// TIA Portal V15.1 export
// export: Created 2024-06-21T08:41:11.7725682Z, ExportSetting WithDefaults, DisplayName Totally Integrated Automation Portal, DisplayVersion V15.1 Update 5, DisplayName TIA Portal Openness, DisplayVersion V15.1 Update 5, DisplayName SINAMICS Startdrive Advanced, DisplayVersion V15.1, DisplayName G130, G150, S120, S150, SINAMICS MV, S210, DisplayVersion V15.1, DisplayName G110M, G120, G120C, G120D, G120P, DisplayVersion V15.1, DisplayName STEP 7 Professional, DisplayVersion V15.1 Update 5, DisplayName STEP 7 Safety, DisplayVersion V15.1, DisplayName WinCC Professional, DisplayVersion V15.1 Update 5, DisplayName SIMATIC Visualization Architect, DisplayVersion V15.1
FUNCTION_BLOCK "LGBShiftRegLine"   // FB6704, FBD
TITLE = LGBShiftRegLine
{ S7_Optimized_Access := 'TRUE' }
VERSION : 0.1
// stored: AutoNumber false, IsIECCheckEnabled false, IsRetainMemResEnabled false, MemoryReserve 100, SetENOAutomatically False, UDAEnableTagReadback false
   VAR_INPUT
      I_VEMData { ExternalAccessible := 'False'; ExternalVisible := 'False'; ExternalWritable := 'False'} : "VEMData";   // VEMData
      I_EncPlsCntr { ExternalAccessible := 'False'; ExternalVisible := 'False'; ExternalWritable := 'False'} : DInt;   // Encoder pulse counter - value from counter card
      I_LineRunning { ExternalAccessible := 'False'; ExternalVisible := 'False'; ExternalWritable := 'False'} : Bool;   // Line running - signal from freq. convertor
      I_TriggerDet { ExternalAccessible := 'False'; ExternalVisible := 'False'; ExternalWritable := 'False'} : Bool;   // Trigger sensor
   END_VAR
   VAR_OUTPUT
      O_SetpBodyPitch { ExternalAccessible := 'False'; ExternalVisible := 'False'; ExternalWritable := 'False'} : Int;   // Setpoint Body pitch (cm)
      O_SetpCycleTime { ExternalAccessible := 'False'; ExternalVisible := 'False'; ExternalWritable := 'False'} : Int;   // Setpoint Cycle time (sec)
      O_SetpSpeed { ExternalAccessible := 'False'; ExternalVisible := 'False'; ExternalWritable := 'False'} : Real;   // Setpoint Speed (m/min)
      O_LineIsEmpty { ExternalAccessible := 'False'; ExternalVisible := 'False'; ExternalWritable := 'False'} : Bool;   // Line is empty
      O_Area1 { ExternalAccessible := 'False'; ExternalVisible := 'False'; ExternalWritable := 'False'} : Bool;   // Position active in the Area
      O_Area2 { ExternalAccessible := 'False'; ExternalVisible := 'False'; ExternalWritable := 'False'} : Bool;   // Position active in the Area
      O_Area3 { ExternalAccessible := 'False'; ExternalVisible := 'False'; ExternalWritable := 'False'} : Bool;   // Position active in the Area
      O_Area4 { ExternalAccessible := 'False'; ExternalVisible := 'False'; ExternalWritable := 'False'} : Bool;   // Position active in the Area
      O_Area5 { ExternalAccessible := 'False'; ExternalVisible := 'False'; ExternalWritable := 'False'} : Bool;   // Position active in the Area
      O_Area6 { ExternalAccessible := 'False'; ExternalVisible := 'False'; ExternalWritable := 'False'} : Bool;   // Position active in the Area
      O_Area7 { ExternalAccessible := 'False'; ExternalVisible := 'False'; ExternalWritable := 'False'} : Bool;   // Position active in the Area
      O_Area8 { ExternalAccessible := 'False'; ExternalVisible := 'False'; ExternalWritable := 'False'} : Bool;   // Position active in the Area
      O_Area9 { ExternalAccessible := 'False'; ExternalVisible := 'False'; ExternalWritable := 'False'} : Bool;   // Position active in the Area
      O_Area10 { ExternalAccessible := 'False'; ExternalVisible := 'False'; ExternalWritable := 'False'} : Bool;   // Position active in the Area
      O_AlarmABCondition { ExternalAccessible := 'False'; ExternalVisible := 'False'; ExternalWritable := 'False'} : Bool;   // Alarm AB Condition
      O_AlarmA { ExternalAccessible := 'False'; ExternalVisible := 'False'; ExternalWritable := 'False'} : Bool;   // Alarm A
      O_AlarmB { ExternalAccessible := 'False'; ExternalVisible := 'False'; ExternalWritable := 'False'} : Bool;   // Alarm B
      O_AlarmC { ExternalAccessible := 'False'; ExternalVisible := 'False'; ExternalWritable := 'False'} : Bool;   // Alarm C
      O_AlarmD { ExternalAccessible := 'False'; ExternalVisible := 'False'; ExternalWritable := 'False'} : Bool;   // Alarm D
      H_AlarmDWord { ExternalAccessible := 'False'; ExternalVisible := 'False'; ExternalWritable := 'False'} : DWord;   // Alarm Word
   END_VAR
   VAR_IN_OUT
      IO_ShiftRegData : "ShiftRegData";   // Line data
      IO_Modes : "Modes";   // Modes
      H_HMI : "H_HMI";   // Animation
      H_GBShiftRegLine : "H_GBShiftRegLine";   // Animation
      C_Config : "ShiftRegLineConfig";   // Config
   END_VAR
   VAR
      AA_EncoderMinMax { ExternalAccessible := 'False'; ExternalVisible := 'False'; ExternalWritable := 'False'} : Bool;   // Settings Min. and Max. range for the encoder is not ok --- Max. must be > Min. and Max. <> 0
      AA_SetpointBodyPitch { ExternalAccessible := 'False'; ExternalVisible := 'False'; ExternalWritable := 'False'} : Bool;   // Setpoint Bodypitch is not ok --- Setpoint must be > 100 cm
      AA_SetpointCycleTime { ExternalAccessible := 'False'; ExternalVisible := 'False'; ExternalWritable := 'False'} : Bool;   // Setpoint CycleTime is not ok --- Setpoint must be > 10 sec
      AA_NbrOfWorkZones { ExternalAccessible := 'False'; ExternalVisible := 'False'; ExternalWritable := 'False'} : Bool;   // Number of work zones is not ok --- Must be >= 2 and <= 30
      AA_EncoderPuls { ExternalAccessible := 'False'; ExternalVisible := 'False'; ExternalWritable := 'False'} : Bool;   // The line is running buth there are no encoder pulses
      AC_Calibration { ExternalAccessible := 'False'; ExternalVisible := 'False'; ExternalWritable := 'False'} : Bool;   // Calibration is not ok. Let the line run and start the calibration
      AC_Area1 { ExternalAccessible := 'False'; ExternalVisible := 'False'; ExternalWritable := 'False'} : Bool;   // Start or End value is not ok Area 1
      AC_Area2 { ExternalAccessible := 'False'; ExternalVisible := 'False'; ExternalWritable := 'False'} : Bool;   // Start or End value is not ok Area 2
      AC_Area3 { ExternalAccessible := 'False'; ExternalVisible := 'False'; ExternalWritable := 'False'} : Bool;   // Start or End value is not ok Area 3
      AC_Area4 { ExternalAccessible := 'False'; ExternalVisible := 'False'; ExternalWritable := 'False'} : Bool;   // Start or End value is not ok Area 4
      AC_Area5 { ExternalAccessible := 'False'; ExternalVisible := 'False'; ExternalWritable := 'False'} : Bool;   // Start or End value is not ok Area 5
      AC_Area6 { ExternalAccessible := 'False'; ExternalVisible := 'False'; ExternalWritable := 'False'} : Bool;   // Start or End value is not ok Area 6
      AC_Area7 { ExternalAccessible := 'False'; ExternalVisible := 'False'; ExternalWritable := 'False'} : Bool;   // Start or End value is not ok Area 7
      AC_Area8 { ExternalAccessible := 'False'; ExternalVisible := 'False'; ExternalWritable := 'False'} : Bool;   // Start or End value is not ok Area 8
      AC_Area9 { ExternalAccessible := 'False'; ExternalVisible := 'False'; ExternalWritable := 'False'} : Bool;   // Start or End value is not ok Area 9
      AC_Area10 { ExternalAccessible := 'False'; ExternalVisible := 'False'; ExternalWritable := 'False'} : Bool;   // Start or End value is not ok Area 10
      AlarmA { ExternalAccessible := 'False'; ExternalVisible := 'False'; ExternalWritable := 'False'} : Bool;   // Alarm A
      AlarmB { ExternalAccessible := 'False'; ExternalVisible := 'False'; ExternalWritable := 'False'} : Bool;   // Alarm B
      AlarmC { ExternalAccessible := 'False'; ExternalVisible := 'False'; ExternalWritable := 'False'} : Bool;   // Alarm C
      AlarmD { ExternalAccessible := 'False'; ExternalVisible := 'False'; ExternalWritable := 'False'} : Bool;   // Alarm D
      AlarmABCondition { ExternalAccessible := 'False'; ExternalVisible := 'False'; ExternalWritable := 'False'} : Bool;   // Alarm AB Condition
      _ShiftRegLineSub { ExternalAccessible := 'False'; ExternalVisible := 'False'; ExternalWritable := 'False'} : "LGBShiftRegLineSub";
   END_VAR
   VAR_TEMP   // added for the SCL form of the ladder/FBD networks
      _w1 : Bool;
   END_VAR
BEGIN

REGION Network 1: **** 7.1 - Submodule - Non-Machine **** Shift Register
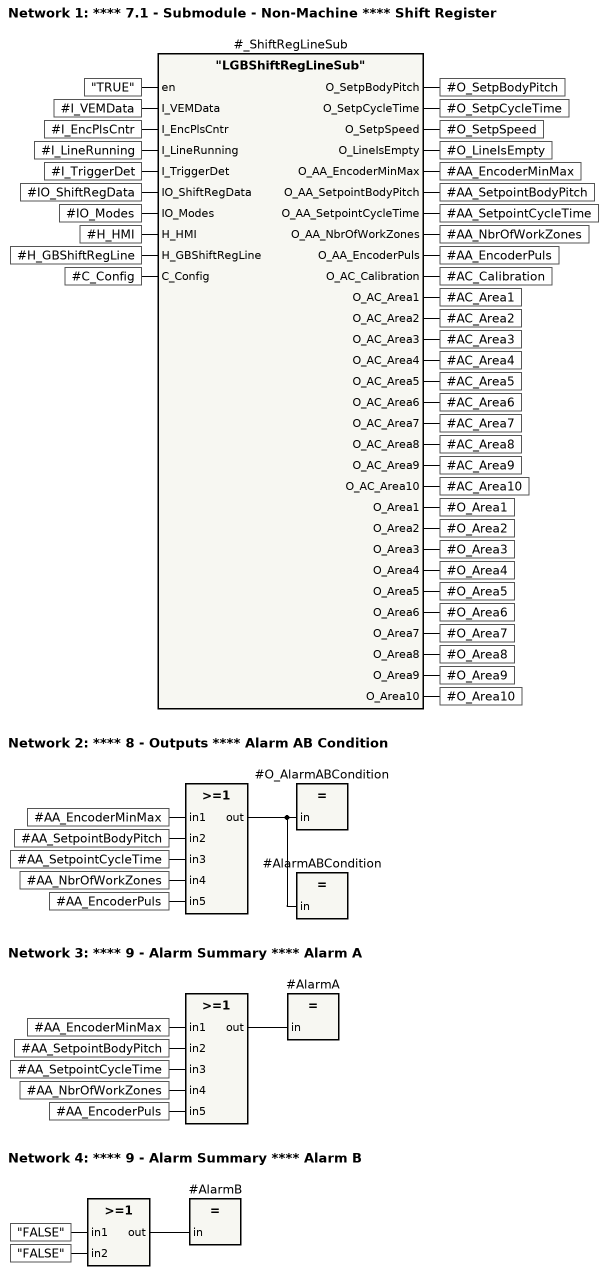
   IF "TRUE" THEN
       #_ShiftRegLineSub(I_VEMData := #I_VEMData,   // "LGBShiftRegLineSub"
                         I_EncPlsCntr := #I_EncPlsCntr,
                         I_LineRunning := #I_LineRunning,
                         I_TriggerDet := #I_TriggerDet,
                         IO_ShiftRegData := #IO_ShiftRegData,
                         IO_Modes := #IO_Modes,
                         H_HMI := #H_HMI,
                         H_GBShiftRegLine := #H_GBShiftRegLine,
                         C_Config := #C_Config,
                         O_SetpBodyPitch => #O_SetpBodyPitch,
                         O_SetpCycleTime => #O_SetpCycleTime,
                         O_SetpSpeed => #O_SetpSpeed,
                         O_LineIsEmpty => #O_LineIsEmpty,
                         O_AA_EncoderMinMax => #AA_EncoderMinMax,
                         O_AA_SetpointBodyPitch => #AA_SetpointBodyPitch,
                         O_AA_SetpointCycleTime => #AA_SetpointCycleTime,
                         O_AA_NbrOfWorkZones => #AA_NbrOfWorkZones,
                         O_AA_EncoderPuls => #AA_EncoderPuls,
                         O_AC_Calibration => #AC_Calibration,
                         O_AC_Area1 => #AC_Area1,
                         O_AC_Area2 => #AC_Area2,
                         O_AC_Area3 => #AC_Area3,
                         O_AC_Area4 => #AC_Area4,
                         O_AC_Area5 => #AC_Area5,
                         O_AC_Area6 => #AC_Area6,
                         O_AC_Area7 => #AC_Area7,
                         O_AC_Area8 => #AC_Area8,
                         O_AC_Area9 => #AC_Area9,
                         O_AC_Area10 => #AC_Area10,
                         O_Area1 => #O_Area1,
                         O_Area2 => #O_Area2,
                         O_Area3 => #O_Area3,
                         O_Area4 => #O_Area4,
                         O_Area5 => #O_Area5,
                         O_Area6 => #O_Area6,
                         O_Area7 => #O_Area7,
                         O_Area8 => #O_Area8,
                         O_Area9 => #O_Area9,
                         O_Area10 => #O_Area10);
   END_IF;
END_REGION

REGION Network 2: **** 8 - Outputs **** Alarm AB Condition
   // Alarm AB Condition
   #O_AlarmABCondition := #AA_EncoderMinMax OR #AA_SetpointBodyPitch OR #AA_SetpointCycleTime OR #AA_NbrOfWorkZones OR #AA_EncoderPuls;
   #AlarmABCondition := #O_AlarmABCondition;
END_REGION

REGION Network 3: **** 9 - Alarm Summary **** Alarm A
   // Alarm A
   #AlarmA := #AA_EncoderMinMax OR #AA_SetpointBodyPitch OR #AA_SetpointCycleTime OR #AA_NbrOfWorkZones OR #AA_EncoderPuls;
END_REGION

REGION Network 4: **** 9 - Alarm Summary **** Alarm B
   // Alarm B
   #AlarmB := "FALSE" OR "FALSE";
END_REGION

REGION Network 5: **** 9 - Alarm Summary **** Alarm C
   // Alarm C
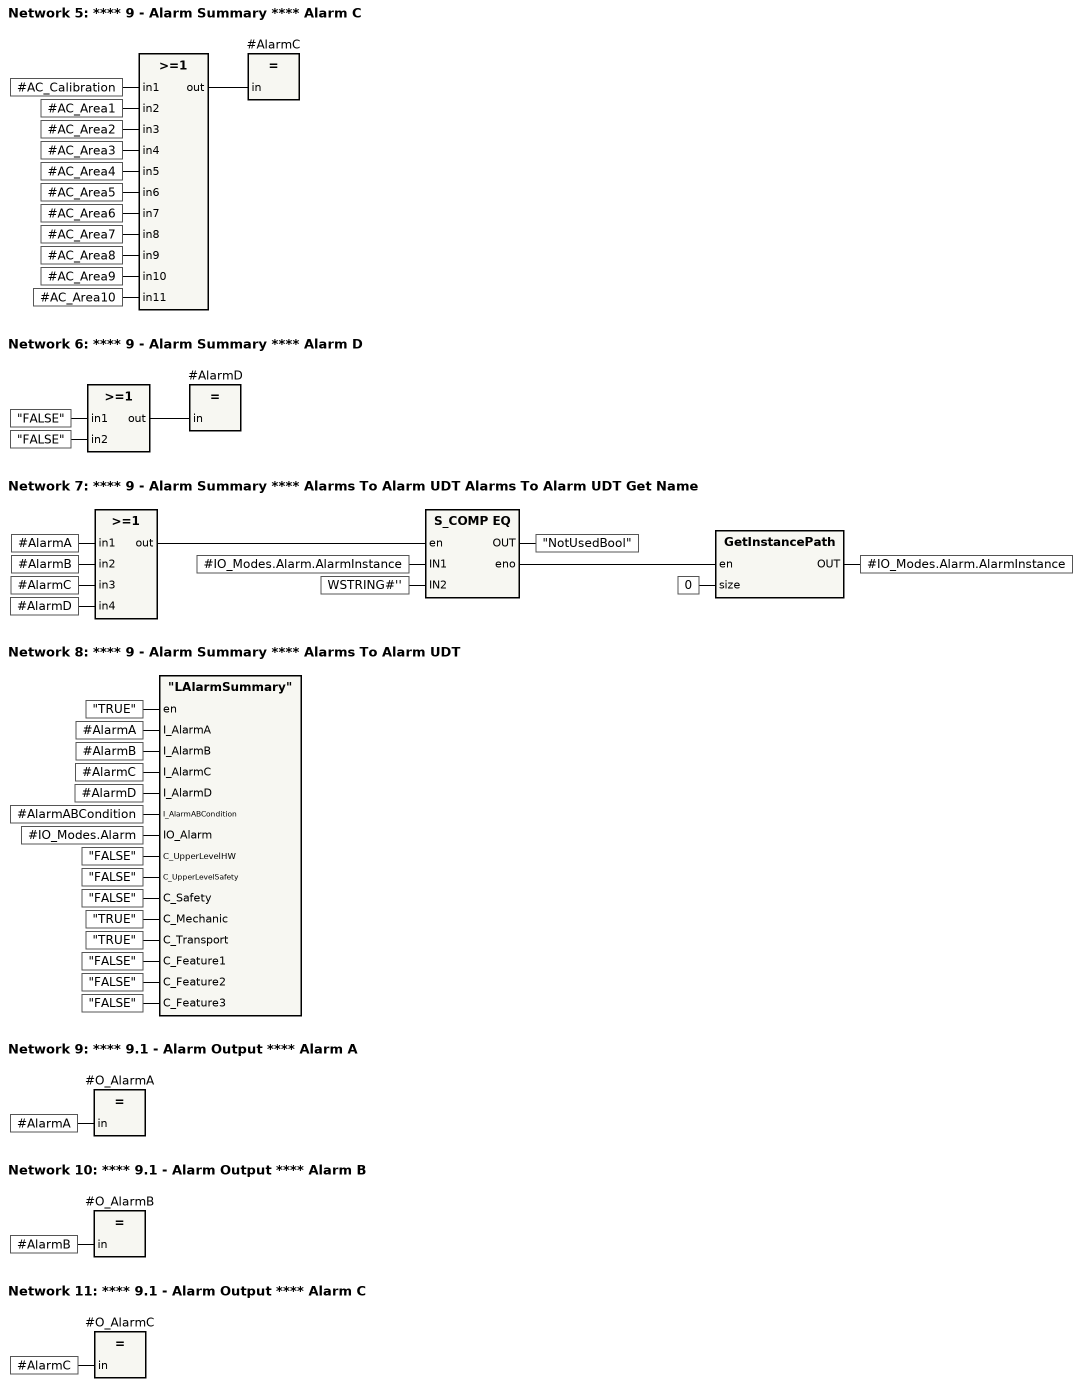
   #AlarmC := #AC_Calibration OR #AC_Area1 OR #AC_Area2 OR #AC_Area3 OR #AC_Area4 OR #AC_Area5 OR #AC_Area6 OR #AC_Area7 OR #AC_Area8 OR #AC_Area9 OR #AC_Area10;
END_REGION

REGION Network 6: **** 9 - Alarm Summary **** Alarm D
   // Alarm D
   #AlarmD := "FALSE" OR "FALSE";
END_REGION

REGION Network 7: **** 9 - Alarm Summary **** Alarms To Alarm UDT Alarms To Alarm UDT Get Name
   // Alarm / Alarm D
   S_COMP(EN := #AlarmA OR #AlarmB OR #AlarmC OR #AlarmD,
          IN1 := #IO_Modes.Alarm.AlarmInstance,
          IN2 := WSTRING#'',
          OUT => "NotUsedBool",
          ENO => #_w1);
   IF #_w1 THEN GetInstancePath(size := 0, OUT => #IO_Modes.Alarm.AlarmInstance); END_IF;
END_REGION

REGION Network 8: **** 9 - Alarm Summary **** Alarms To Alarm UDT
   // Alarm / Alarm D
   IF "TRUE" THEN
       "LAlarmSummary"(I_AlarmA := #AlarmA,
                       I_AlarmB := #AlarmB,
                       I_AlarmC := #AlarmC,
                       I_AlarmD := #AlarmD,
                       I_AlarmABCondition := #AlarmABCondition,
                       IO_Alarm := #IO_Modes.Alarm,
                       C_UpperLevelHW := "FALSE",
                       C_UpperLevelSafety := "FALSE",
                       C_Safety := "FALSE",
                       C_Mechanic := "TRUE",
                       C_Transport := "TRUE",
                       C_Feature1 := "FALSE",
                       C_Feature2 := "FALSE",
                       C_Feature3 := "FALSE");
   END_IF;
END_REGION

REGION Network 9: **** 9.1 - Alarm Output **** Alarm A
   // Alarm A
   #O_AlarmA := #AlarmA;
END_REGION

REGION Network 10: **** 9.1 - Alarm Output **** Alarm B
   // Alarm B
   #O_AlarmB := #AlarmB;
END_REGION

REGION Network 11: **** 9.1 - Alarm Output **** Alarm C
   // Alarm C
   #O_AlarmC := #AlarmC;
END_REGION

REGION Network 12: **** 9.1 - Alarm Output **** Alarm D
   // Alarm D
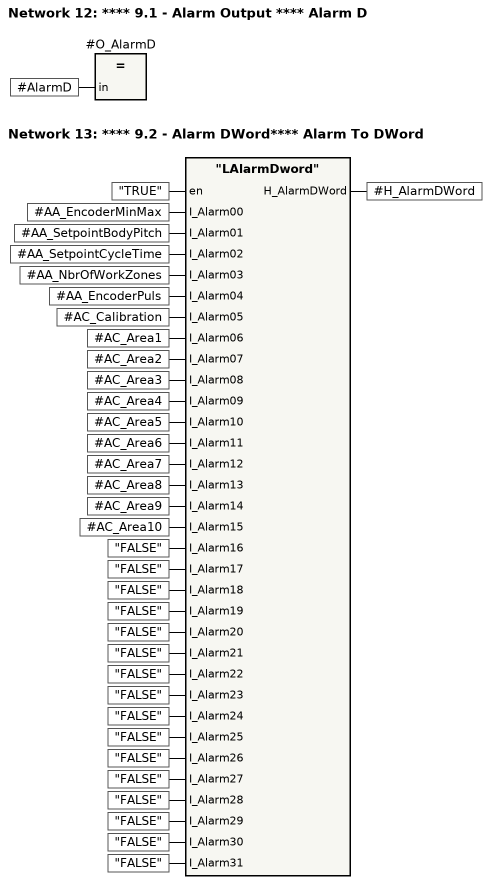
   #O_AlarmD := #AlarmD;
END_REGION

REGION Network 13: **** 9.2 - Alarm DWord**** Alarm To DWord
   // Alarm To DWord
   IF "TRUE" THEN
       "LAlarmDword"(I_Alarm00 := #AA_EncoderMinMax,
                     I_Alarm01 := #AA_SetpointBodyPitch,
                     I_Alarm02 := #AA_SetpointCycleTime,
                     I_Alarm03 := #AA_NbrOfWorkZones,
                     I_Alarm04 := #AA_EncoderPuls,
                     I_Alarm05 := #AC_Calibration,
                     I_Alarm06 := #AC_Area1,
                     I_Alarm07 := #AC_Area2,
                     I_Alarm08 := #AC_Area3,
                     I_Alarm09 := #AC_Area4,
                     I_Alarm10 := #AC_Area5,
                     I_Alarm11 := #AC_Area6,
                     I_Alarm12 := #AC_Area7,
                     I_Alarm13 := #AC_Area8,
                     I_Alarm14 := #AC_Area9,
                     I_Alarm15 := #AC_Area10,
                     I_Alarm16 := "FALSE",
                     I_Alarm17 := "FALSE",
                     I_Alarm18 := "FALSE",
                     I_Alarm19 := "FALSE",
                     I_Alarm20 := "FALSE",
                     I_Alarm21 := "FALSE",
                     I_Alarm22 := "FALSE",
                     I_Alarm23 := "FALSE",
                     I_Alarm24 := "FALSE",
                     I_Alarm25 := "FALSE",
                     I_Alarm26 := "FALSE",
                     I_Alarm27 := "FALSE",
                     I_Alarm28 := "FALSE",
                     I_Alarm29 := "FALSE",
                     I_Alarm30 := "FALSE",
                     I_Alarm31 := "FALSE",
                     H_AlarmDWord => #H_AlarmDWord);
   END_IF;
END_REGION
END_FUNCTION_BLOCK
